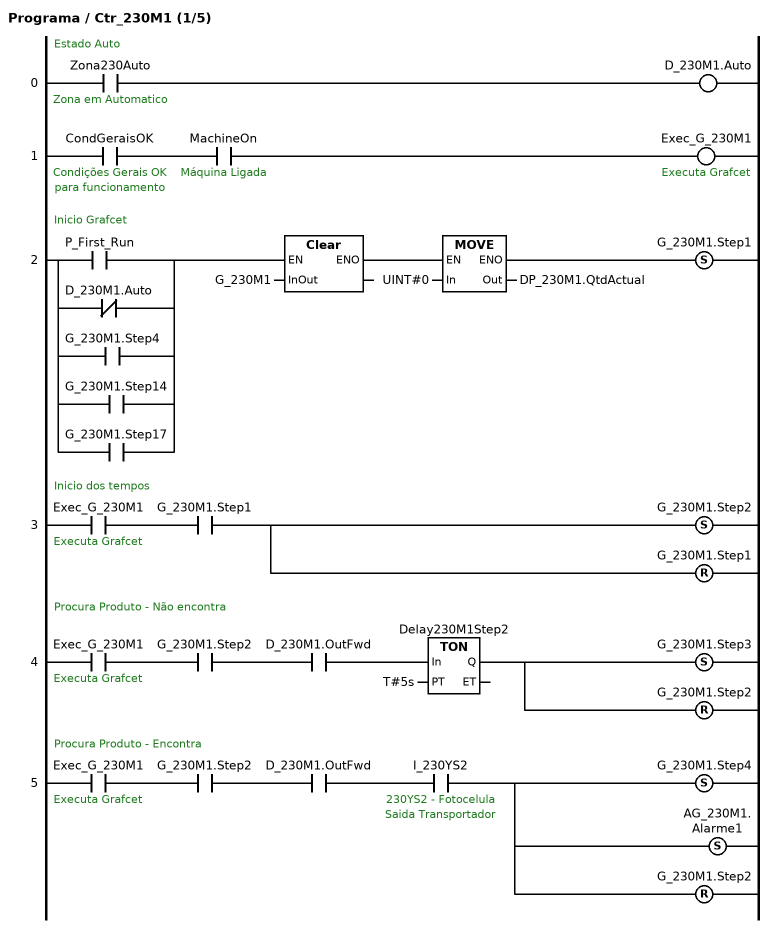
(* [picture p72: Programa / Ctr_230M1, rungs 0-5] *)
(* Rung 0: Estado Auto *)
D_230M1.Auto := Zona230Auto;
(* Rung 1 *)
Exec_G_230M1 := CondGeraisOK AND MachineOn;
(* Rung 2: Inicio Grafcet *)
_p131 := P_First_Run OR NOT D_230M1.Auto OR G_230M1.Step4 OR G_230M1.Step14 OR G_230M1.Step17;
IF _p131 THEN
    Clear(InOut := G_230M1);
    DP_230M1.QtdActual := UINT#0;
    G_230M1.Step1 := TRUE;
END_IF;
(* Rung 3: Inicio dos tempos *)
_p132 := Exec_G_230M1 AND G_230M1.Step1;
IF _p132 THEN
    G_230M1.Step2 := TRUE;
    G_230M1.Step1 := FALSE;
END_IF;
(* Rung 4: Procura Produto - Não encontra *)
Delay230M1Step2(In := Exec_G_230M1 AND G_230M1.Step2 AND D_230M1.OutFwd, PT := T#5s);
IF Delay230M1Step2.Q THEN
    G_230M1.Step3 := TRUE;
    G_230M1.Step2 := FALSE;
END_IF;
(* Rung 5: Procura Produto - Encontra *)
_p133 := Exec_G_230M1 AND G_230M1.Step2 AND D_230M1.OutFwd AND I_230YS2;
IF _p133 THEN
    G_230M1.Step4 := TRUE;
    AG_230M1.Alarme1 := TRUE;
    G_230M1.Step2 := FALSE;
END_IF;

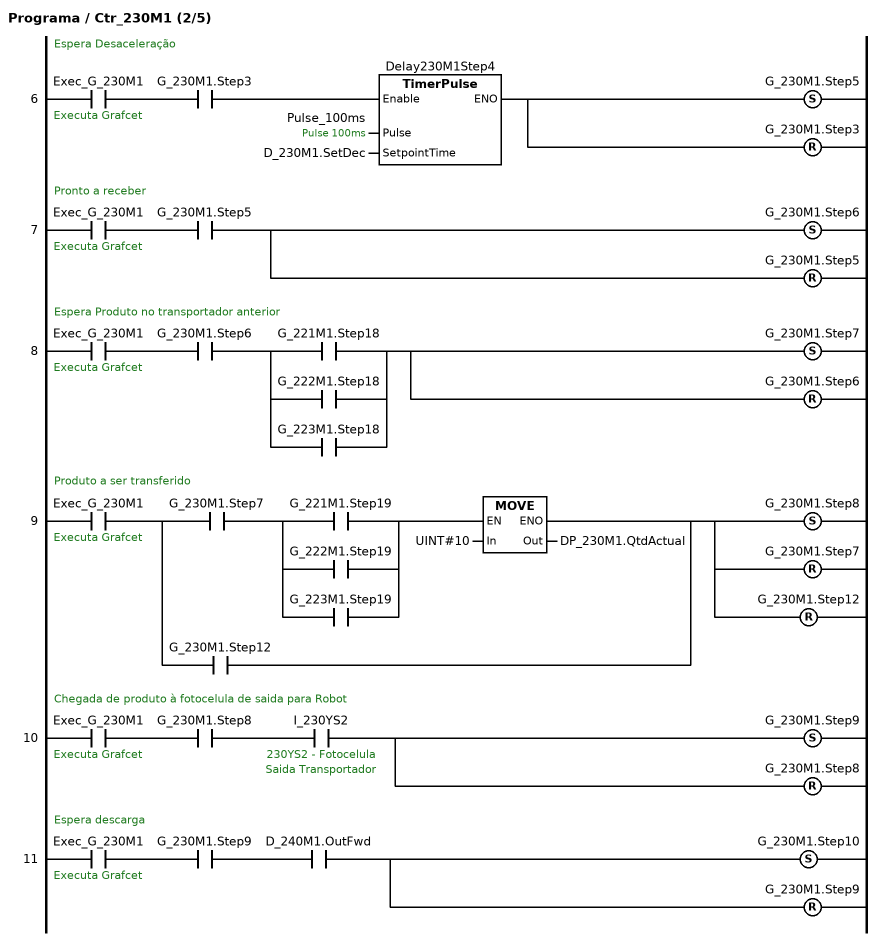
(* Rung 6: Espera Desaceleração *)
Delay230M1Step4(Enable := Exec_G_230M1 AND G_230M1.Step3, Pulse := Pulse_100ms, SetpointTime := D_230M1.SetDec);
IF Delay230M1Step4.ENO THEN
    G_230M1.Step5 := TRUE;
    G_230M1.Step3 := FALSE;
END_IF;
(* Rung 7: Pronto a receber *)
_p134 := Exec_G_230M1 AND G_230M1.Step5;
IF _p134 THEN
    G_230M1.Step6 := TRUE;
    G_230M1.Step5 := FALSE;
END_IF;
(* Rung 8: Espera Produto no transportador anterior *)
_p135 := Exec_G_230M1 AND G_230M1.Step6 AND (G_221M1.Step18 OR G_222M1.Step18 OR G_223M1.Step18);
IF _p135 THEN
    G_230M1.Step7 := TRUE;
    G_230M1.Step6 := FALSE;
END_IF;
(* Rung 9: Produto a ser transferido *)
IF Exec_G_230M1 AND G_230M1.Step7 AND (G_221M1.Step19 OR G_222M1.Step19 OR G_223M1.Step19) THEN
    DP_230M1.QtdActual := UINT#10;
END_IF;
_p136 := Exec_G_230M1 AND ((G_230M1.Step7 AND (G_221M1.Step19 OR G_222M1.Step19 OR G_223M1.Step19)) OR G_230M1.Step12);
IF _p136 THEN
    G_230M1.Step8 := TRUE;
    G_230M1.Step7 := FALSE;
    G_230M1.Step12 := FALSE;
END_IF;
(* Rung 10: Chegada de produto à fotocelula de saida para Robot *)
_p137 := Exec_G_230M1 AND G_230M1.Step8 AND I_230YS2;
IF _p137 THEN
    G_230M1.Step9 := TRUE;
    G_230M1.Step8 := FALSE;
END_IF;
(* Rung 11: Espera descarga *)
_p138 := Exec_G_230M1 AND G_230M1.Step9 AND D_240M1.OutFwd;
IF _p138 THEN
    G_230M1.Step10 := TRUE;
    G_230M1.Step9 := FALSE;
END_IF;

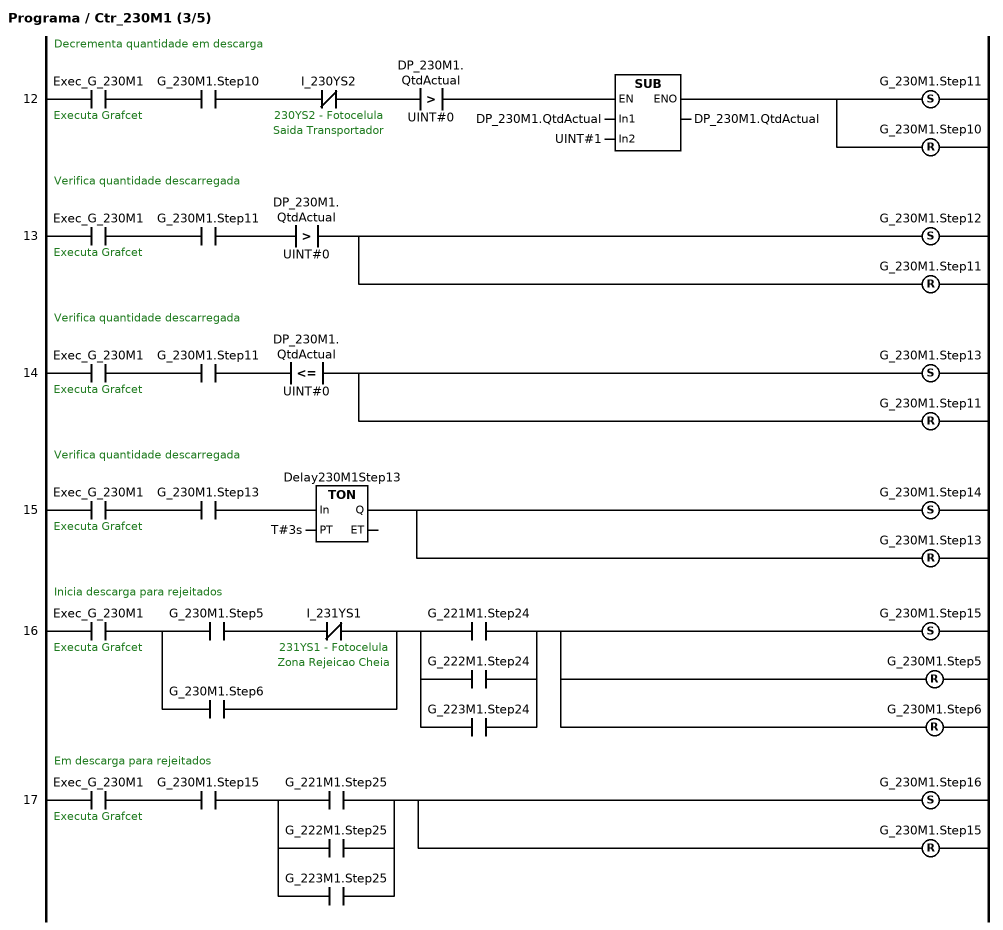
(* Rung 12: Decrementa quantidade em descarga *)
_p139 := Exec_G_230M1 AND G_230M1.Step10 AND NOT I_230YS2 AND (DP_230M1.QtdActual > UINT#0);
IF _p139 THEN
    DP_230M1.QtdActual := DP_230M1.QtdActual - UINT#1;
    G_230M1.Step11 := TRUE;
    G_230M1.Step10 := FALSE;
END_IF;
(* Rung 13: Verifica quantidade descarregada *)
_p140 := Exec_G_230M1 AND G_230M1.Step11 AND (DP_230M1.QtdActual > UINT#0);
IF _p140 THEN
    G_230M1.Step12 := TRUE;
    G_230M1.Step11 := FALSE;
END_IF;
(* Rung 14: Verifica quantidade descarregada *)
_p141 := Exec_G_230M1 AND G_230M1.Step11 AND (DP_230M1.QtdActual <= UINT#0);
IF _p141 THEN
    G_230M1.Step13 := TRUE;
    G_230M1.Step11 := FALSE;
END_IF;
(* Rung 15: Verifica quantidade descarregada *)
Delay230M1Step13(In := Exec_G_230M1 AND G_230M1.Step13, PT := T#3s);
IF Delay230M1Step13.Q THEN
    G_230M1.Step14 := TRUE;
    G_230M1.Step13 := FALSE;
END_IF;
(* Rung 16: Inicia descarga para rejeitados *)
_p142 := Exec_G_230M1 AND ((G_230M1.Step5 AND NOT I_231YS1) OR G_230M1.Step6) AND (G_221M1.Step24 OR G_222M1.Step24 OR G_223M1.Step24);
IF _p142 THEN
    G_230M1.Step15 := TRUE;
    G_230M1.Step5 := FALSE;
    G_230M1.Step6 := FALSE;
END_IF;
(* Rung 17: Em descarga para rejeitados *)
_p143 := Exec_G_230M1 AND G_230M1.Step15 AND (G_221M1.Step25 OR G_222M1.Step25 OR G_223M1.Step25);
IF _p143 THEN
    G_230M1.Step16 := TRUE;
    G_230M1.Step15 := FALSE;
END_IF;

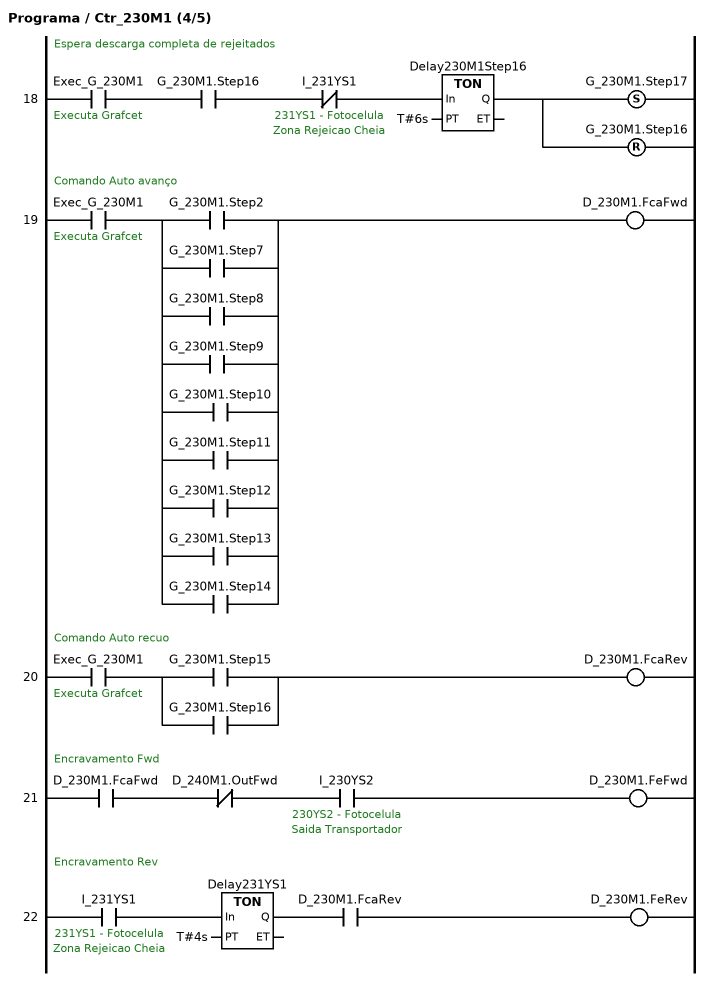
(* Rung 18: Espera descarga completa de rejeitados *)
Delay230M1Step16(In := Exec_G_230M1 AND G_230M1.Step16 AND NOT I_231YS1, PT := T#6s);
IF Delay230M1Step16.Q THEN
    G_230M1.Step17 := TRUE;
    G_230M1.Step16 := FALSE;
END_IF;
(* Rung 19: Comando Auto avanço *)
D_230M1.FcaFwd := Exec_G_230M1 AND (G_230M1.Step2 OR G_230M1.Step7 OR G_230M1.Step8 OR G_230M1.Step9 OR G_230M1.Step10 OR G_230M1.Step11 OR G_230M1.Step12 OR G_230M1.Step13 OR G_230M1.Step14);
(* Rung 20: Comando Auto recuo *)
D_230M1.FcaRev := Exec_G_230M1 AND (G_230M1.Step15 OR G_230M1.Step16);
(* Rung 21: Encravamento Fwd *)
D_230M1.FeFwd := D_230M1.FcaFwd AND NOT D_240M1.OutFwd AND I_230YS2;
(* Rung 22: Encravamento Rev *)
Delay231YS1(In := I_231YS1, PT := T#4s);
D_230M1.FeRev := Delay231YS1.Q AND D_230M1.FcaRev;

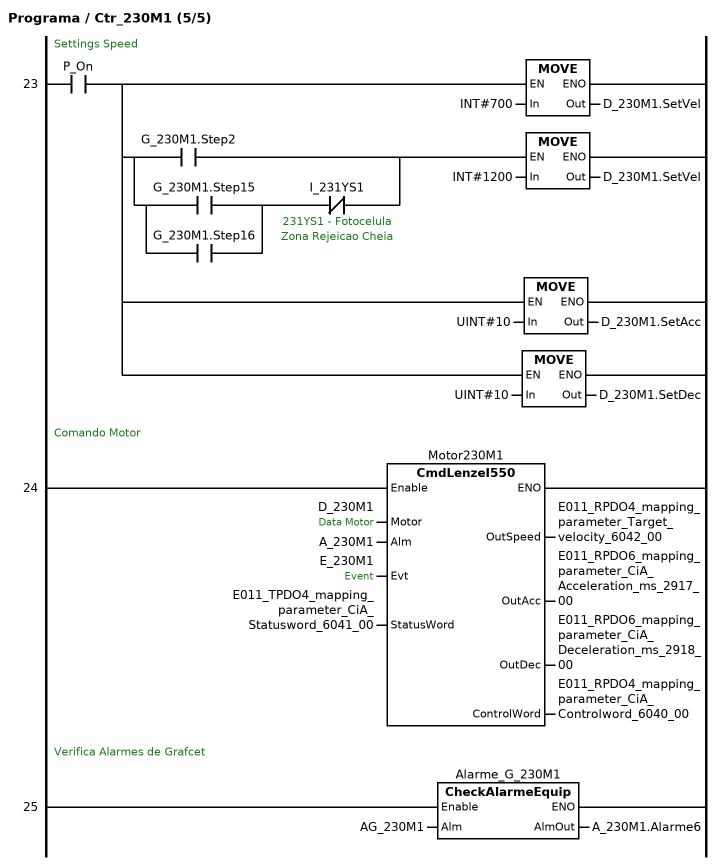
(* Rung 23: Settings Speed *)
IF P_On THEN D_230M1.SetVel := INT#700; END_IF;
IF P_On AND (G_230M1.Step2 OR ((G_230M1.Step15 OR G_230M1.Step16) AND NOT I_231YS1)) THEN
    D_230M1.SetVel := INT#1200;
END_IF;
IF P_On THEN
    D_230M1.SetAcc := UINT#10;
    D_230M1.SetDec := UINT#10;
END_IF;
(* Rung 24: Comando Motor *)
Motor230M1(Enable := TRUE, Motor := D_230M1, Alm := A_230M1, Evt := E_230M1, StatusWord := E011_TPDO4_mapping_parameter_CiA_Statusword_6041_00, OutSpeed => E011_RPDO4_mapping_parameter_Target_velocity_6042_00, OutAcc => E011_RPDO6_mapping_parameter_CiA_Acceleration_ms_2917_00, OutDec => E011_RPDO6_mapping_parameter_CiA_Deceleration_ms_2918_00, ControlWord => E011_RPDO4_mapping_parameter_CiA_Controlword_6040_00);
(* Rung 25: Verifica Alarmes de Grafcet *)
Alarme_G_230M1(Enable := TRUE, Alm := AG_230M1, AlmOut => A_230M1.Alarme6);

(* Section Ctr_240M1: ladder, written here as Structured Text *)

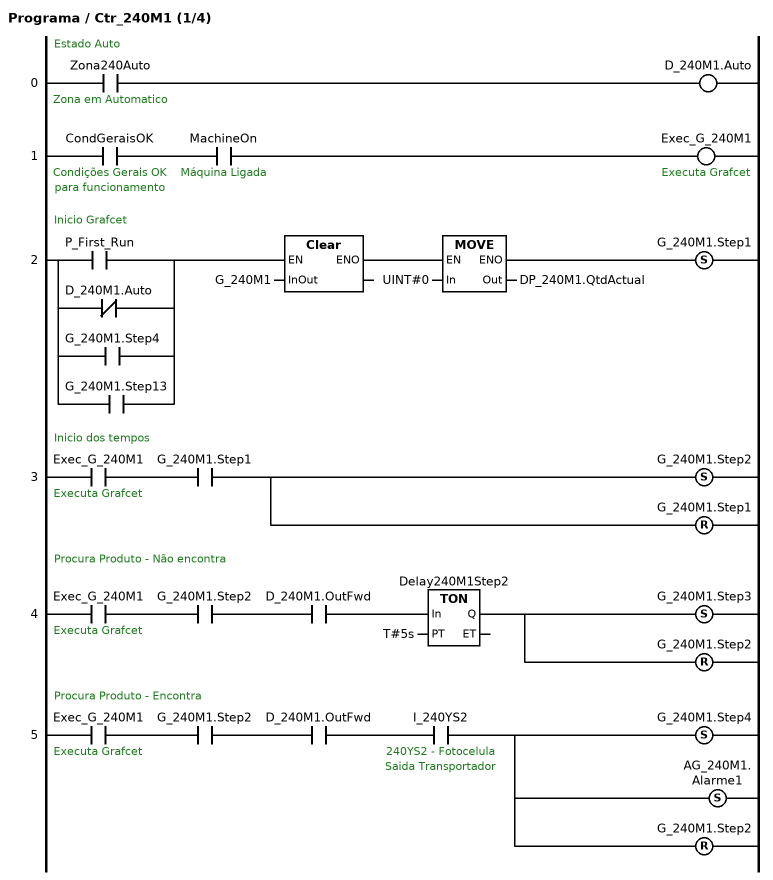
(* Rung 0: Estado Auto *)
D_240M1.Auto := Zona240Auto;
(* Rung 1 *)
Exec_G_240M1 := CondGeraisOK AND MachineOn;
(* Rung 2: Inicio Grafcet *)
_p144 := P_First_Run OR NOT D_240M1.Auto OR G_240M1.Step4 OR G_240M1.Step13;
IF _p144 THEN
    Clear(InOut := G_240M1);
    DP_240M1.QtdActual := UINT#0;
    G_240M1.Step1 := TRUE;
END_IF;
(* Rung 3: Inicio dos tempos *)
_p145 := Exec_G_240M1 AND G_240M1.Step1;
IF _p145 THEN
    G_240M1.Step2 := TRUE;
    G_240M1.Step1 := FALSE;
END_IF;
(* Rung 4: Procura Produto - Não encontra *)
Delay240M1Step2(In := Exec_G_240M1 AND G_240M1.Step2 AND D_240M1.OutFwd, PT := T#5s);
IF Delay240M1Step2.Q THEN
    G_240M1.Step3 := TRUE;
    G_240M1.Step2 := FALSE;
END_IF;
(* Rung 5: Procura Produto - Encontra *)
_p146 := Exec_G_240M1 AND G_240M1.Step2 AND D_240M1.OutFwd AND I_240YS2;
IF _p146 THEN
    G_240M1.Step4 := TRUE;
    AG_240M1.Alarme1 := TRUE;
    G_240M1.Step2 := FALSE;
END_IF;

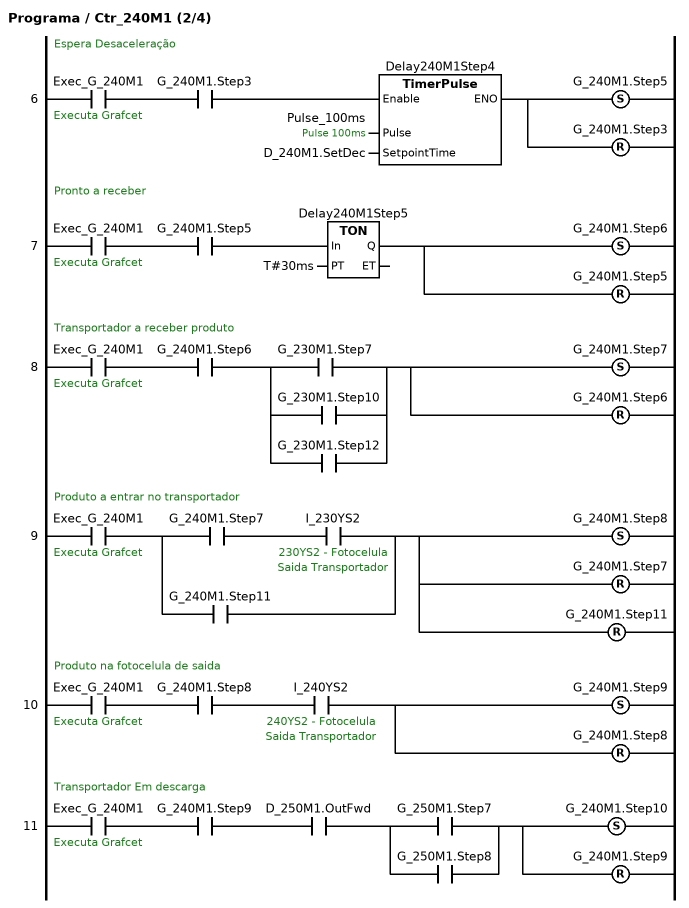
(* Rung 6: Espera Desaceleração *)
Delay240M1Step4(Enable := Exec_G_240M1 AND G_240M1.Step3, Pulse := Pulse_100ms, SetpointTime := D_240M1.SetDec);
IF Delay240M1Step4.ENO THEN
    G_240M1.Step5 := TRUE;
    G_240M1.Step3 := FALSE;
END_IF;
(* Rung 7: Pronto a receber *)
Delay240M1Step5(In := Exec_G_240M1 AND G_240M1.Step5, PT := T#30ms);
IF Delay240M1Step5.Q THEN
    G_240M1.Step6 := TRUE;
    G_240M1.Step5 := FALSE;
END_IF;
(* Rung 8: Transportador a receber produto *)
_p147 := Exec_G_240M1 AND G_240M1.Step6 AND (G_230M1.Step7 OR G_230M1.Step10 OR G_230M1.Step12);
IF _p147 THEN
    G_240M1.Step7 := TRUE;
    G_240M1.Step6 := FALSE;
END_IF;
(* Rung 9: Produto a entrar no transportador *)
_p148 := Exec_G_240M1 AND ((G_240M1.Step7 AND I_230YS2) OR G_240M1.Step11);
IF _p148 THEN
    G_240M1.Step8 := TRUE;
    G_240M1.Step7 := FALSE;
    G_240M1.Step11 := FALSE;
END_IF;
(* Rung 10: Produto na fotocelula de saida *)
_p149 := Exec_G_240M1 AND G_240M1.Step8 AND I_240YS2;
IF _p149 THEN
    G_240M1.Step9 := TRUE;
    G_240M1.Step8 := FALSE;
END_IF;
(* Rung 11: Transportador Em descarga *)
_p150 := Exec_G_240M1 AND G_240M1.Step9 AND D_250M1.OutFwd AND (G_250M1.Step7 OR G_250M1.Step8);
IF _p150 THEN
    G_240M1.Step10 := TRUE;
    G_240M1.Step9 := FALSE;
END_IF;

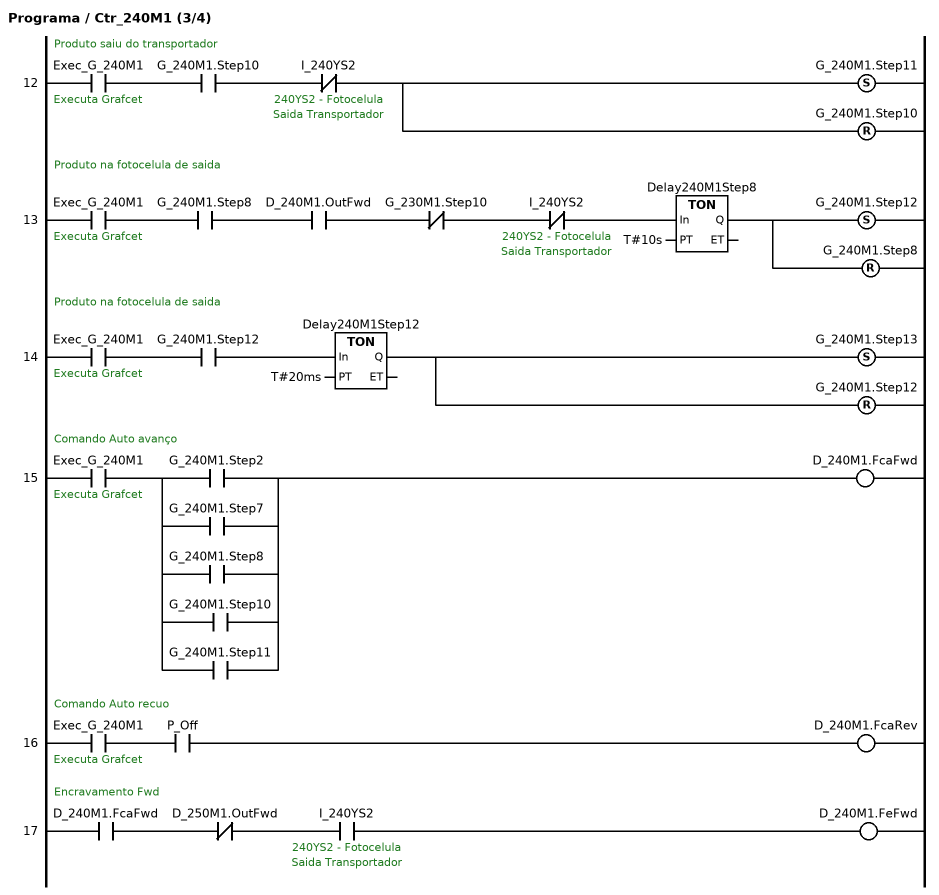
(* Rung 12: Produto saiu do transportador *)
_p151 := Exec_G_240M1 AND G_240M1.Step10 AND NOT I_240YS2;
IF _p151 THEN
    G_240M1.Step11 := TRUE;
    G_240M1.Step10 := FALSE;
END_IF;
(* Rung 13: Produto na fotocelula de saida *)
Delay240M1Step8(In := Exec_G_240M1 AND G_240M1.Step8 AND D_240M1.OutFwd AND NOT G_230M1.Step10 AND NOT I_240YS2, PT := T#10s);
IF Delay240M1Step8.Q THEN
    G_240M1.Step12 := TRUE;
    G_240M1.Step8 := FALSE;
END_IF;
(* Rung 14: Produto na fotocelula de saida *)
Delay240M1Step12(In := Exec_G_240M1 AND G_240M1.Step12, PT := T#20ms);
IF Delay240M1Step12.Q THEN
    G_240M1.Step13 := TRUE;
    G_240M1.Step12 := FALSE;
END_IF;
(* Rung 15: Comando Auto avanço *)
D_240M1.FcaFwd := Exec_G_240M1 AND (G_240M1.Step2 OR G_240M1.Step7 OR G_240M1.Step8 OR G_240M1.Step10 OR G_240M1.Step11);
(* Rung 16: Comando Auto recuo *)
D_240M1.FcaRev := Exec_G_240M1 AND P_Off;
(* Rung 17: Encravamento Fwd *)
D_240M1.FeFwd := D_240M1.FcaFwd AND NOT D_250M1.OutFwd AND I_240YS2;

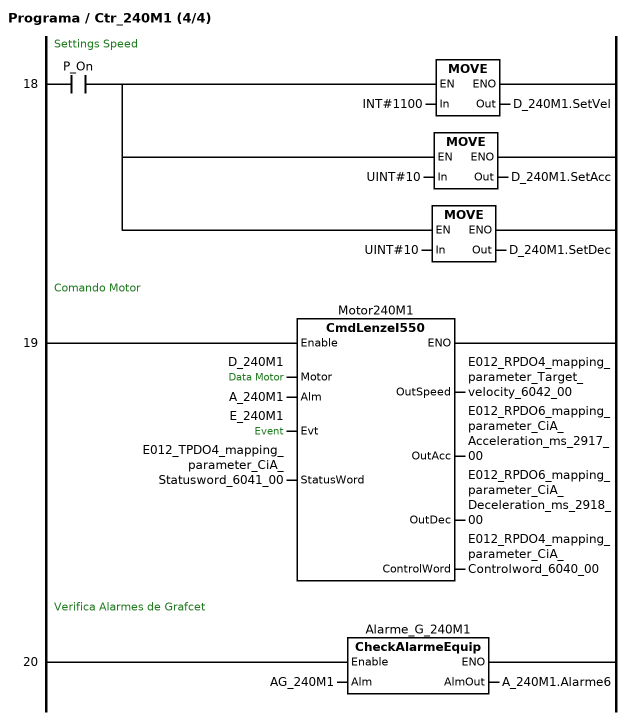
(* Rung 18: Settings Speed *)
IF P_On THEN
    D_240M1.SetVel := INT#1100;
    D_240M1.SetAcc := UINT#10;
    D_240M1.SetDec := UINT#10;
END_IF;
(* Rung 19: Comando Motor *)
Motor240M1(Enable := TRUE, Motor := D_240M1, Alm := A_240M1, Evt := E_240M1, StatusWord := E012_TPDO4_mapping_parameter_CiA_Statusword_6041_00, OutSpeed => E012_RPDO4_mapping_parameter_Target_velocity_6042_00, OutAcc => E012_RPDO6_mapping_parameter_CiA_Acceleration_ms_2917_00, OutDec => E012_RPDO6_mapping_parameter_CiA_Deceleration_ms_2918_00, ControlWord => E012_RPDO4_mapping_parameter_CiA_Controlword_6040_00);
(* Rung 20: Verifica Alarmes de Grafcet *)
Alarme_G_240M1(Enable := TRUE, Alm := AG_240M1, AlmOut => A_240M1.Alarme6);

(* Section Ctr_250M1: ladder, written here as Structured Text *)

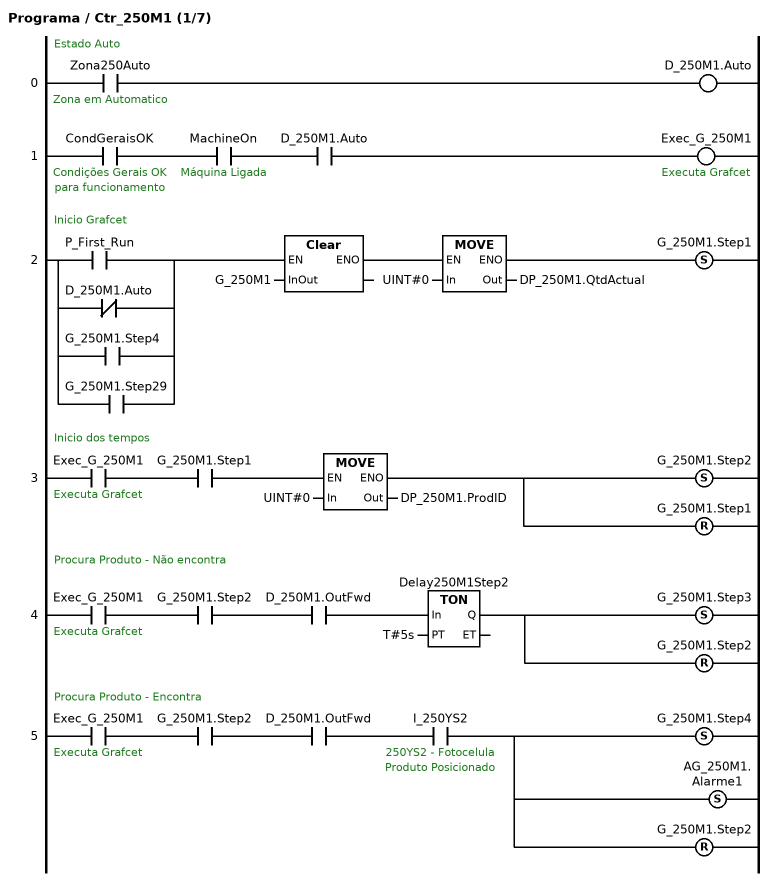
(* Rung 0: Estado Auto *)
D_250M1.Auto := Zona250Auto;
(* Rung 1 *)
Exec_G_250M1 := CondGeraisOK AND MachineOn AND D_250M1.Auto;
(* Rung 2: Inicio Grafcet *)
_p152 := P_First_Run OR NOT D_250M1.Auto OR G_250M1.Step4 OR G_250M1.Step29;
IF _p152 THEN
    Clear(InOut := G_250M1);
    DP_250M1.QtdActual := UINT#0;
    G_250M1.Step1 := TRUE;
END_IF;
(* Rung 3: Inicio dos tempos *)
IF Exec_G_250M1 AND G_250M1.Step1 THEN DP_250M1.ProdID := UINT#0; END_IF;
_p153 := Exec_G_250M1 AND G_250M1.Step1;
IF _p153 THEN
    G_250M1.Step2 := TRUE;
    G_250M1.Step1 := FALSE;
END_IF;
(* Rung 4: Procura Produto - Não encontra *)
Delay250M1Step2(In := Exec_G_250M1 AND G_250M1.Step2 AND D_250M1.OutFwd, PT := T#5s);
IF Delay250M1Step2.Q THEN
    G_250M1.Step3 := TRUE;
    G_250M1.Step2 := FALSE;
END_IF;
(* Rung 5: Procura Produto - Encontra *)
_p154 := Exec_G_250M1 AND G_250M1.Step2 AND D_250M1.OutFwd AND I_250YS2;
IF _p154 THEN
    G_250M1.Step4 := TRUE;
    AG_250M1.Alarme1 := TRUE;
    G_250M1.Step2 := FALSE;
END_IF;

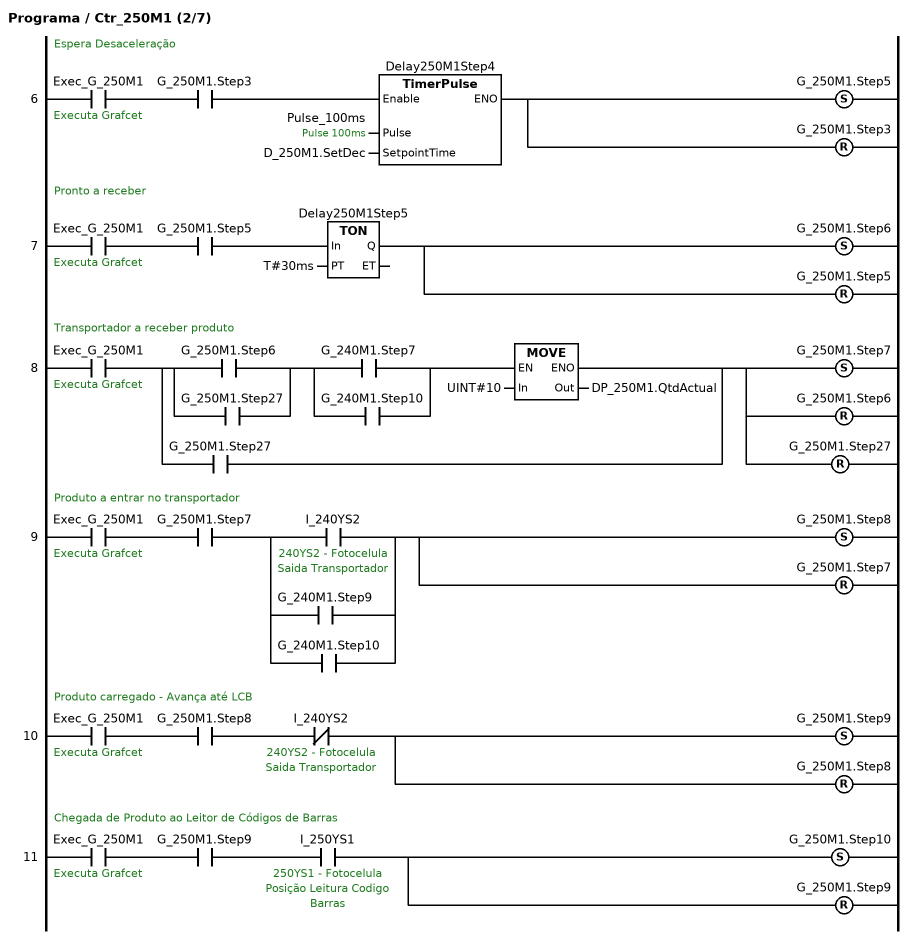
(* Rung 6: Espera Desaceleração *)
Delay250M1Step4(Enable := Exec_G_250M1 AND G_250M1.Step3, Pulse := Pulse_100ms, SetpointTime := D_250M1.SetDec);
IF Delay250M1Step4.ENO THEN
    G_250M1.Step5 := TRUE;
    G_250M1.Step3 := FALSE;
END_IF;
(* Rung 7: Pronto a receber *)
Delay250M1Step5(In := Exec_G_250M1 AND G_250M1.Step5, PT := T#30ms);
IF Delay250M1Step5.Q THEN
    G_250M1.Step6 := TRUE;
    G_250M1.Step5 := FALSE;
END_IF;
(* Rung 8: Transportador a receber produto *)
IF Exec_G_250M1 AND (G_250M1.Step6 OR G_250M1.Step27) AND (G_240M1.Step7 OR G_240M1.Step10) THEN
    DP_250M1.QtdActual := UINT#10;
END_IF;
_p155 := Exec_G_250M1 AND (((G_250M1.Step6 OR G_250M1.Step27) AND (G_240M1.Step7 OR G_240M1.Step10)) OR G_250M1.Step27);
IF _p155 THEN
    G_250M1.Step7 := TRUE;
    G_250M1.Step6 := FALSE;
    G_250M1.Step27 := FALSE;
END_IF;
(* Rung 9: Produto a entrar no transportador *)
_p156 := Exec_G_250M1 AND G_250M1.Step7 AND (I_240YS2 OR G_240M1.Step9 OR G_240M1.Step10);
IF _p156 THEN
    G_250M1.Step8 := TRUE;
    G_250M1.Step7 := FALSE;
END_IF;
(* Rung 10: Produto carregado - Avança até LCB *)
_p157 := Exec_G_250M1 AND G_250M1.Step8 AND NOT I_240YS2;
IF _p157 THEN
    G_250M1.Step9 := TRUE;
    G_250M1.Step8 := FALSE;
END_IF;
(* Rung 11: Chegada de Produto ao Leitor de Códigos de Barras *)
_p158 := Exec_G_250M1 AND G_250M1.Step9 AND I_250YS1;
IF _p158 THEN
    G_250M1.Step10 := TRUE;
    G_250M1.Step9 := FALSE;
END_IF;

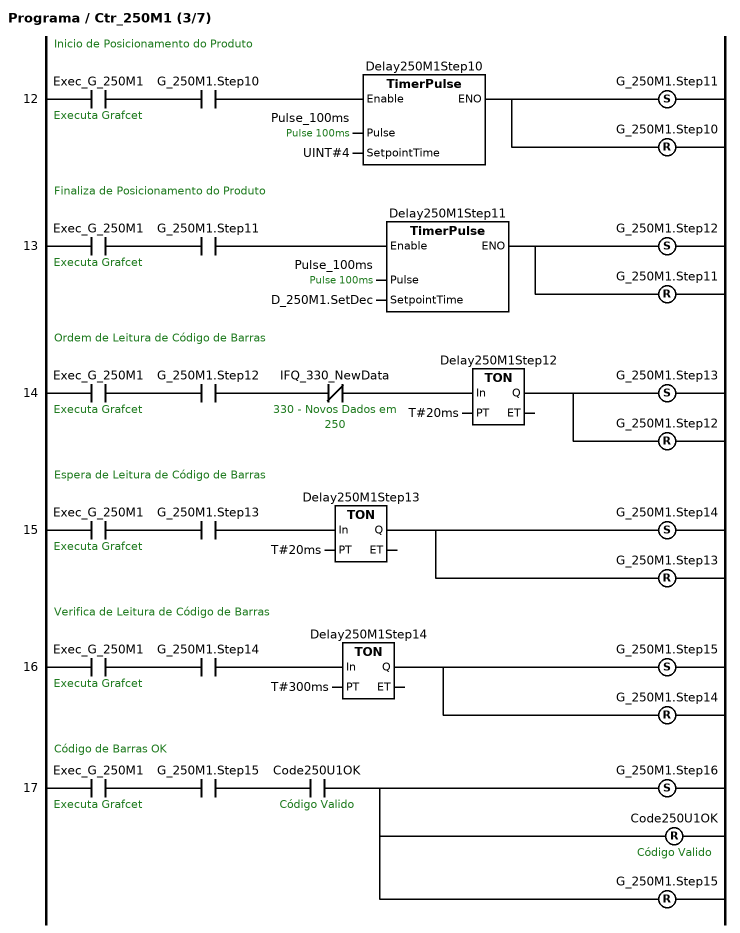
(* Rung 12: Inicio de Posicionamento do Produto *)
Delay250M1Step10(Enable := Exec_G_250M1 AND G_250M1.Step10, Pulse := Pulse_100ms, SetpointTime := UINT#4);
IF Delay250M1Step10.ENO THEN
    G_250M1.Step11 := TRUE;
    G_250M1.Step10 := FALSE;
END_IF;
(* Rung 13: Finaliza de Posicionamento do Produto *)
Delay250M1Step11(Enable := Exec_G_250M1 AND G_250M1.Step11, Pulse := Pulse_100ms, SetpointTime := D_250M1.SetDec);
IF Delay250M1Step11.ENO THEN
    G_250M1.Step12 := TRUE;
    G_250M1.Step11 := FALSE;
END_IF;
(* Rung 14: Ordem de Leitura de Código de Barras *)
Delay250M1Step12(In := Exec_G_250M1 AND G_250M1.Step12 AND NOT IFQ_330_NewData, PT := T#20ms);
IF Delay250M1Step12.Q THEN
    G_250M1.Step13 := TRUE;
    G_250M1.Step12 := FALSE;
END_IF;
(* Rung 15: Espera de Leitura de Código de Barras *)
Delay250M1Step13(In := Exec_G_250M1 AND G_250M1.Step13, PT := T#20ms);
IF Delay250M1Step13.Q THEN
    G_250M1.Step14 := TRUE;
    G_250M1.Step13 := FALSE;
END_IF;
(* Rung 16: Verifica de Leitura de Código de Barras *)
Delay250M1Step14(In := Exec_G_250M1 AND G_250M1.Step14, PT := T#300ms);
IF Delay250M1Step14.Q THEN
    G_250M1.Step15 := TRUE;
    G_250M1.Step14 := FALSE;
END_IF;
(* Rung 17: Código de Barras OK *)
_p159 := Exec_G_250M1 AND G_250M1.Step15 AND Code250U1OK;
IF _p159 THEN
    G_250M1.Step16 := TRUE;
    Code250U1OK := FALSE;
    G_250M1.Step15 := FALSE;
END_IF;

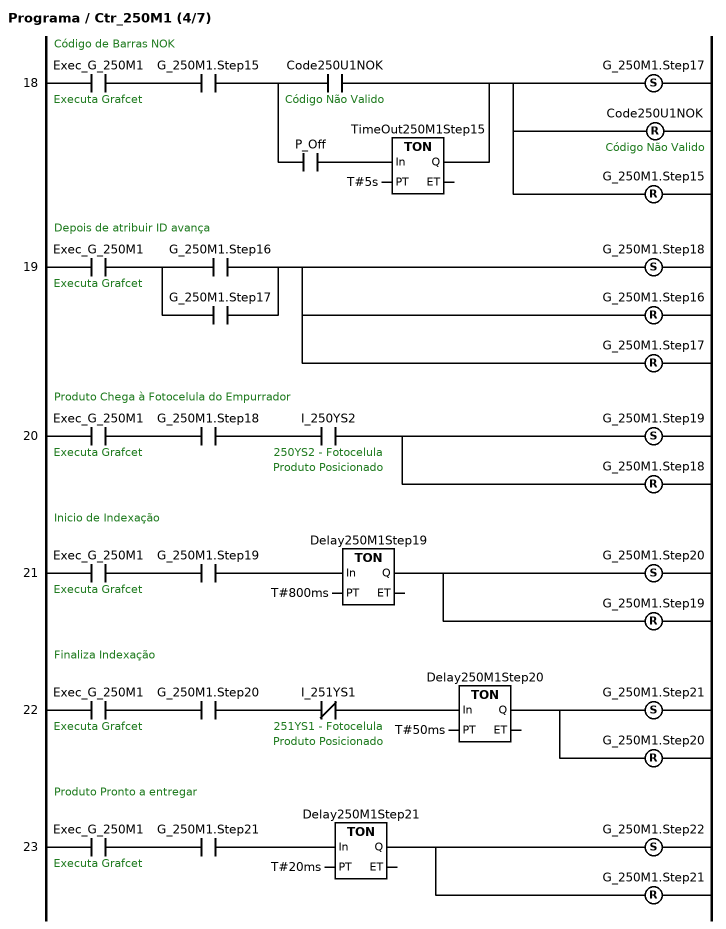
(* Rung 18: Código de Barras NOK *)
TimeOut250M1Step15(In := Exec_G_250M1 AND G_250M1.Step15 AND P_Off, PT := T#5s);
_p160 := (Exec_G_250M1 AND G_250M1.Step15 AND Code250U1NOK) OR TimeOut250M1Step15.Q;
IF _p160 THEN
    G_250M1.Step17 := TRUE;
    Code250U1NOK := FALSE;
    G_250M1.Step15 := FALSE;
END_IF;
(* Rung 19: Depois de atribuir ID avança *)
_p161 := Exec_G_250M1 AND (G_250M1.Step16 OR G_250M1.Step17);
IF _p161 THEN
    G_250M1.Step18 := TRUE;
    G_250M1.Step16 := FALSE;
    G_250M1.Step17 := FALSE;
END_IF;
(* Rung 20: Produto Chega à Fotocelula do Empurrador *)
_p162 := Exec_G_250M1 AND G_250M1.Step18 AND I_250YS2;
IF _p162 THEN
    G_250M1.Step19 := TRUE;
    G_250M1.Step18 := FALSE;
END_IF;
(* Rung 21: Inicio de Indexação *)
Delay250M1Step19(In := Exec_G_250M1 AND G_250M1.Step19, PT := T#800ms);
IF Delay250M1Step19.Q THEN
    G_250M1.Step20 := TRUE;
    G_250M1.Step19 := FALSE;
END_IF;
(* Rung 22: Finaliza Indexação *)
Delay250M1Step20(In := Exec_G_250M1 AND G_250M1.Step20 AND NOT I_251YS1, PT := T#50ms);
IF Delay250M1Step20.Q THEN
    G_250M1.Step21 := TRUE;
    G_250M1.Step20 := FALSE;
END_IF;
(* Rung 23: Produto Pronto a entregar *)
Delay250M1Step21(In := Exec_G_250M1 AND G_250M1.Step21, PT := T#20ms);
IF Delay250M1Step21.Q THEN
    G_250M1.Step22 := TRUE;
    G_250M1.Step21 := FALSE;
END_IF;

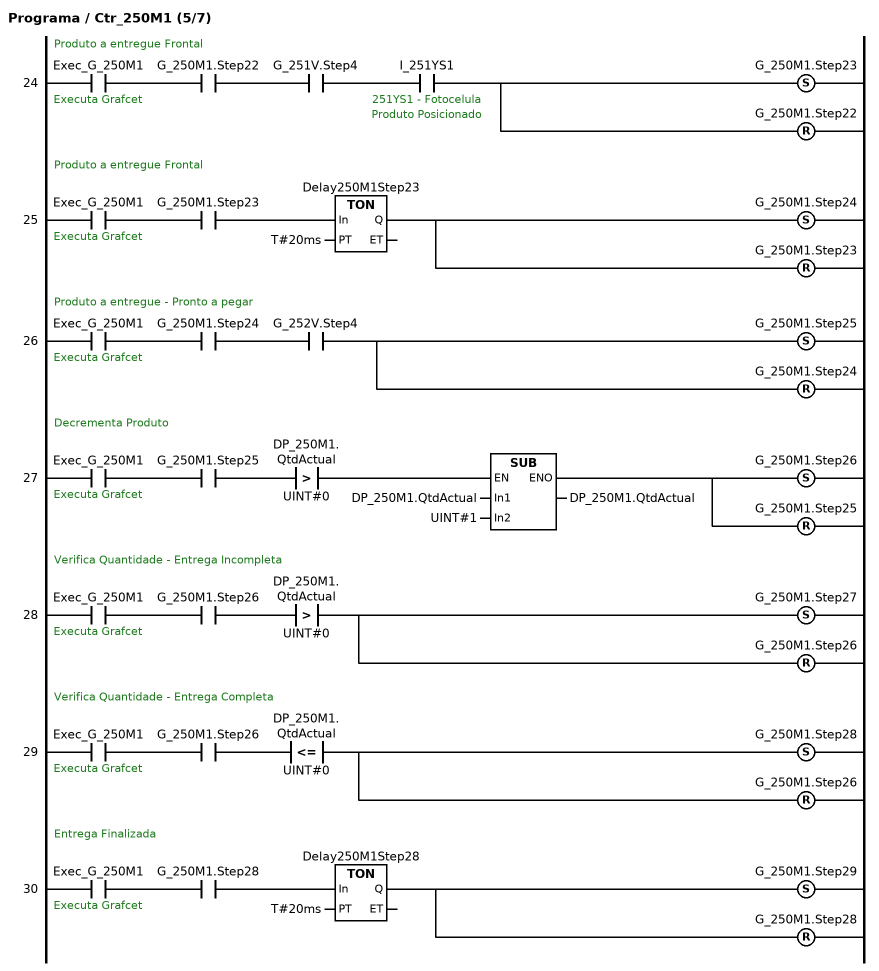
(* Rung 24: Produto a entregue Frontal *)
_p163 := Exec_G_250M1 AND G_250M1.Step22 AND G_251V.Step4 AND I_251YS1;
IF _p163 THEN
    G_250M1.Step23 := TRUE;
    G_250M1.Step22 := FALSE;
END_IF;
(* Rung 25: Produto a entregue Frontal *)
Delay250M1Step23(In := Exec_G_250M1 AND G_250M1.Step23, PT := T#20ms);
IF Delay250M1Step23.Q THEN
    G_250M1.Step24 := TRUE;
    G_250M1.Step23 := FALSE;
END_IF;
(* Rung 26: Produto a entregue - Pronto a pegar *)
_p164 := Exec_G_250M1 AND G_250M1.Step24 AND G_252V.Step4;
IF _p164 THEN
    G_250M1.Step25 := TRUE;
    G_250M1.Step24 := FALSE;
END_IF;
(* Rung 27: Decrementa Produto *)
_p165 := Exec_G_250M1 AND G_250M1.Step25 AND (DP_250M1.QtdActual > UINT#0);
IF _p165 THEN
    DP_250M1.QtdActual := DP_250M1.QtdActual - UINT#1;
    G_250M1.Step26 := TRUE;
    G_250M1.Step25 := FALSE;
END_IF;
(* Rung 28: Verifica Quantidade - Entrega Incompleta *)
_p166 := Exec_G_250M1 AND G_250M1.Step26 AND (DP_250M1.QtdActual > UINT#0);
IF _p166 THEN
    G_250M1.Step27 := TRUE;
    G_250M1.Step26 := FALSE;
END_IF;
(* Rung 29: Verifica Quantidade - Entrega Completa *)
_p167 := Exec_G_250M1 AND G_250M1.Step26 AND (DP_250M1.QtdActual <= UINT#0);
IF _p167 THEN
    G_250M1.Step28 := TRUE;
    G_250M1.Step26 := FALSE;
END_IF;
(* Rung 30: Entrega Finalizada *)
Delay250M1Step28(In := Exec_G_250M1 AND G_250M1.Step28, PT := T#20ms);
IF Delay250M1Step28.Q THEN
    G_250M1.Step29 := TRUE;
    G_250M1.Step28 := FALSE;
END_IF;

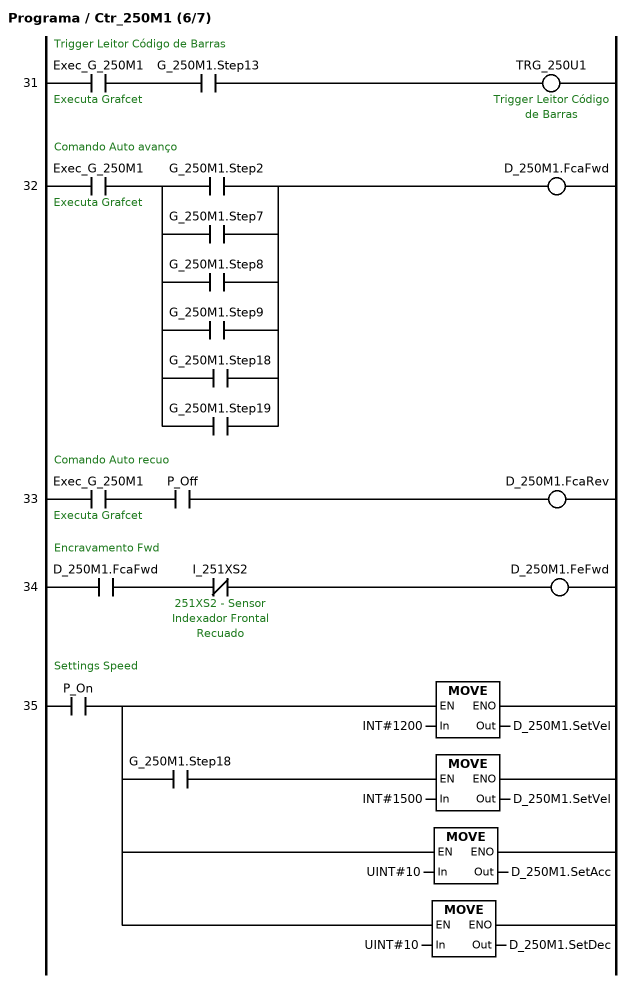
(* Rung 31: Trigger Leitor Código de Barras *)
TRG_250U1 := Exec_G_250M1 AND G_250M1.Step13;
(* Rung 32: Comando Auto avanço *)
D_250M1.FcaFwd := Exec_G_250M1 AND (G_250M1.Step2 OR G_250M1.Step7 OR G_250M1.Step8 OR G_250M1.Step9 OR G_250M1.Step18 OR G_250M1.Step19);
(* Rung 33: Comando Auto recuo *)
D_250M1.FcaRev := Exec_G_250M1 AND P_Off;
(* Rung 34: Encravamento Fwd *)
D_250M1.FeFwd := D_250M1.FcaFwd AND NOT I_251XS2;
(* Rung 35: Settings Speed *)
IF P_On THEN D_250M1.SetVel := INT#1200; END_IF;
IF P_On AND G_250M1.Step18 THEN D_250M1.SetVel := INT#1500; END_IF;
IF P_On THEN
    D_250M1.SetAcc := UINT#10;
    D_250M1.SetDec := UINT#10;
END_IF;

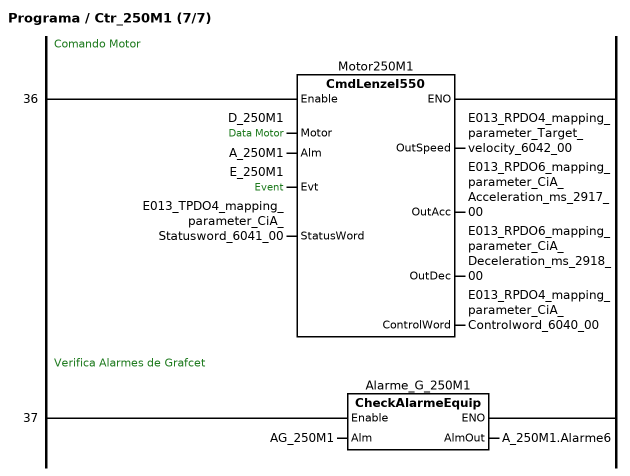
(* Rung 36: Comando Motor *)
Motor250M1(Enable := TRUE, Motor := D_250M1, Alm := A_250M1, Evt := E_250M1, StatusWord := E013_TPDO4_mapping_parameter_CiA_Statusword_6041_00, OutSpeed => E013_RPDO4_mapping_parameter_Target_velocity_6042_00, OutAcc => E013_RPDO6_mapping_parameter_CiA_Acceleration_ms_2917_00, OutDec => E013_RPDO6_mapping_parameter_CiA_Deceleration_ms_2918_00, ControlWord => E013_RPDO4_mapping_parameter_CiA_Controlword_6040_00);
(* Rung 37: Verifica Alarmes de Grafcet *)
Alarme_G_250M1(Enable := TRUE, Alm := AG_250M1, AlmOut => A_250M1.Alarme6);

(* Section Data_250U1: ladder, written here as Structured Text *)

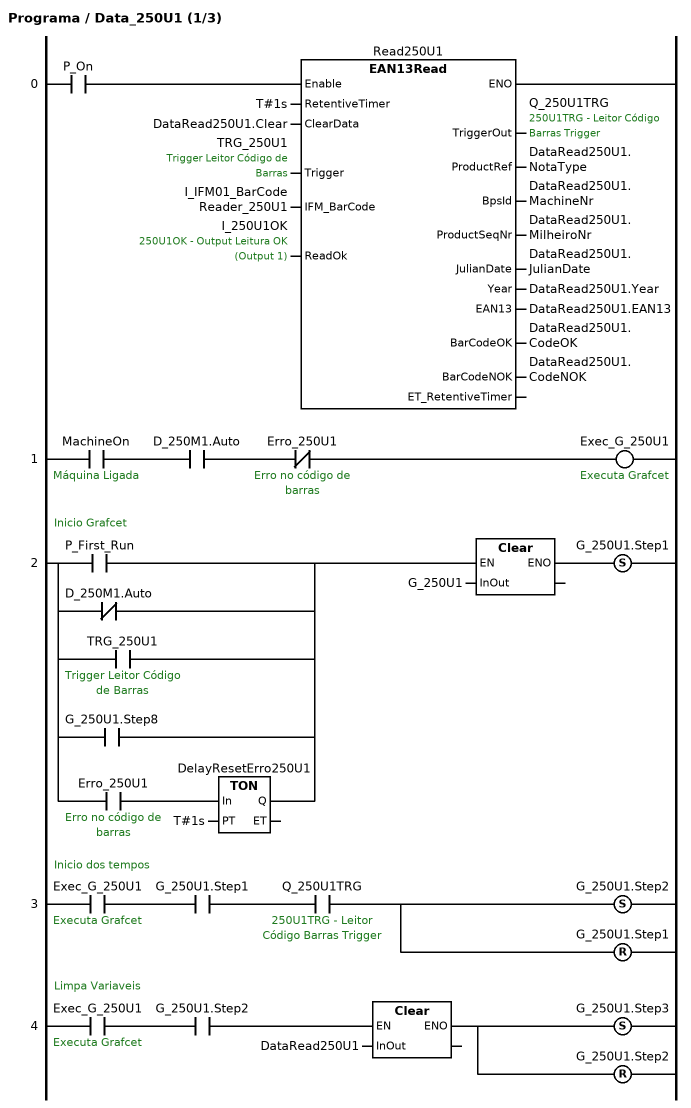
(* Rung 0 *)
Read250U1(Enable := P_On, RetentiveTimer := T#1s, ClearData := DataRead250U1.Clear, Trigger := TRG_250U1, IFM_BarCode := I_IFM01_BarCodeReader_250U1, ReadOk := I_250U1OK, TriggerOut => Q_250U1TRG, ProductRef => DataRead250U1.NotaType, BpsId => DataRead250U1.MachineNr, ProductSeqNr => DataRead250U1.MilheiroNr, JulianDate => DataRead250U1.JulianDate, Year => DataRead250U1.Year, EAN13 => DataRead250U1.EAN13, BarCodeOK => DataRead250U1.CodeOK, BarCodeNOK => DataRead250U1.CodeNOK);
(* Rung 1 *)
Exec_G_250U1 := MachineOn AND D_250M1.Auto AND NOT Erro_250U1;
(* Rung 2: Inicio Grafcet *)
DelayResetErro250U1(In := Erro_250U1, PT := T#1s);
_p168 := P_First_Run OR NOT D_250M1.Auto OR TRG_250U1 OR G_250U1.Step8 OR DelayResetErro250U1.Q;
IF _p168 THEN
    Clear(InOut := G_250U1);
    G_250U1.Step1 := TRUE;
END_IF;
(* Rung 3: Inicio dos tempos *)
_p169 := Exec_G_250U1 AND G_250U1.Step1 AND Q_250U1TRG;
IF _p169 THEN
    G_250U1.Step2 := TRUE;
    G_250U1.Step1 := FALSE;
END_IF;
(* Rung 4: Limpa Variaveis *)
IF Exec_G_250U1 AND G_250U1.Step2 THEN Clear(InOut := DataRead250U1); END_IF;
_p170 := Exec_G_250U1 AND G_250U1.Step2;
IF _p170 THEN
    G_250U1.Step3 := TRUE;
    G_250U1.Step2 := FALSE;
END_IF;

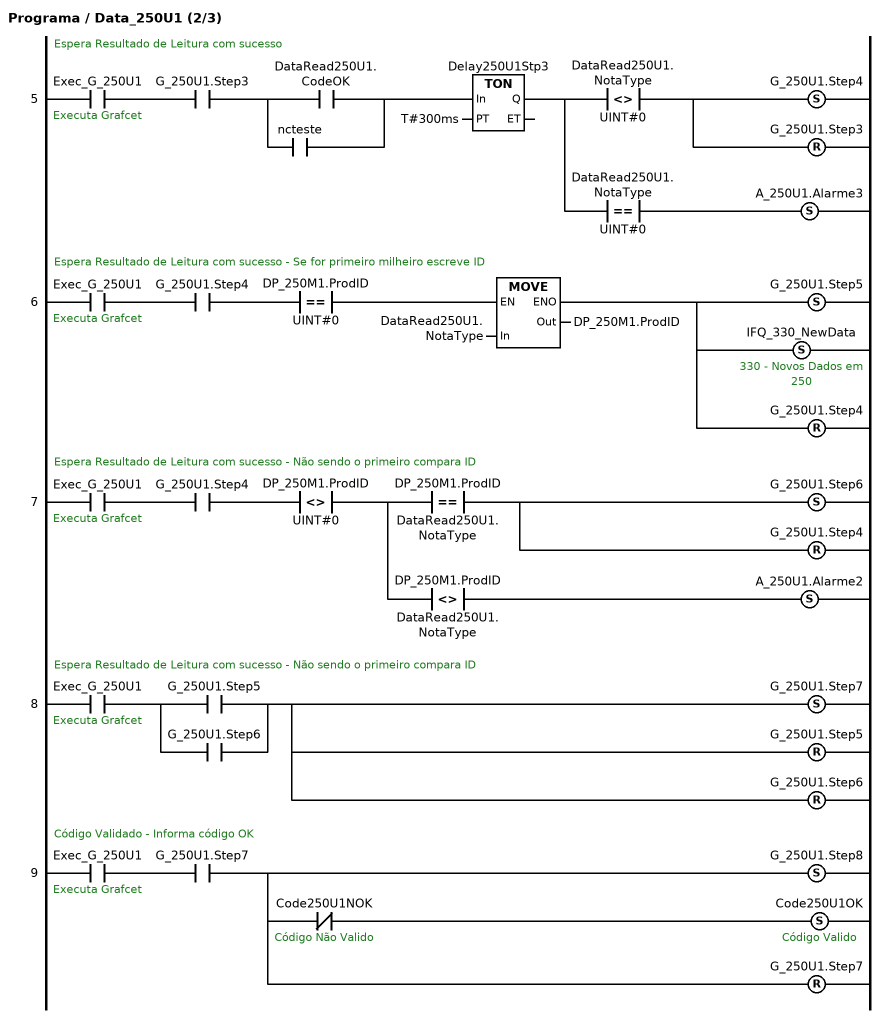
(* Rung 5: Espera Resultado de Leitura com sucesso *)
Delay250U1Stp3(In := Exec_G_250U1 AND G_250U1.Step3 AND (DataRead250U1.CodeOK OR ncteste), PT := T#300ms);
_p171 := Delay250U1Stp3.Q AND (DataRead250U1.NotaType <> UINT#0);
IF _p171 THEN
    G_250U1.Step4 := TRUE;
    G_250U1.Step3 := FALSE;
END_IF;
IF Delay250U1Stp3.Q AND (DataRead250U1.NotaType = UINT#0) THEN A_250U1.Alarme3 := TRUE; END_IF;
(* Rung 6: Espera Resultado de Leitura com sucesso - Se for primeiro milheiro escreve ID *)
_p172 := Exec_G_250U1 AND G_250U1.Step4 AND (DP_250M1.ProdID = UINT#0);
IF _p172 THEN
    DP_250M1.ProdID := DataRead250U1.NotaType;
    G_250U1.Step5 := TRUE;
    IFQ_330_NewData := TRUE;
    G_250U1.Step4 := FALSE;
END_IF;
(* Rung 7: Espera Resultado de Leitura com sucesso - Não sendo o primeiro compara ID *)
_p173 := Exec_G_250U1 AND G_250U1.Step4 AND (DP_250M1.ProdID <> UINT#0);
_p174 := _p173 AND (DP_250M1.ProdID = DataRead250U1.NotaType);
IF _p174 THEN
    G_250U1.Step6 := TRUE;
    G_250U1.Step4 := FALSE;
END_IF;
IF _p173 AND (DP_250M1.ProdID <> DataRead250U1.NotaType) THEN A_250U1.Alarme2 := TRUE; END_IF;
(* Rung 8: Espera Resultado de Leitura com sucesso - Não sendo o primeiro compara ID *)
_p175 := Exec_G_250U1 AND (G_250U1.Step5 OR G_250U1.Step6);
IF _p175 THEN
    G_250U1.Step7 := TRUE;
    G_250U1.Step5 := FALSE;
    G_250U1.Step6 := FALSE;
END_IF;
(* Rung 9: Código Validado - Informa código OK *)
_p176 := Exec_G_250U1 AND G_250U1.Step7;
IF _p176 THEN G_250U1.Step8 := TRUE; END_IF;
IF _p176 AND NOT Code250U1NOK THEN Code250U1OK := TRUE; END_IF;
IF _p176 THEN G_250U1.Step7 := FALSE; END_IF;

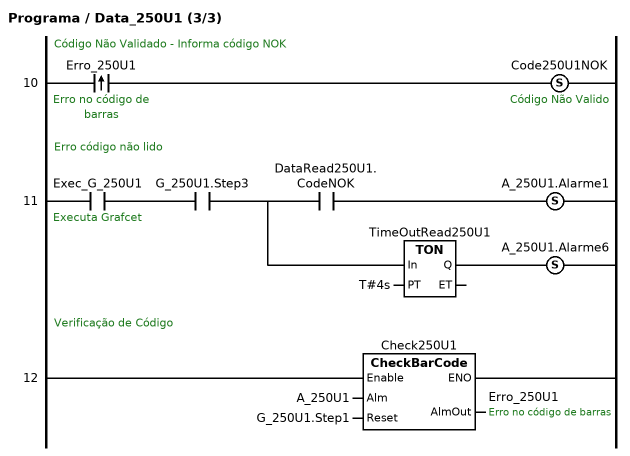
(* Rung 10: Código Não Validado - Informa código NOK *)
_e177(CLK := Erro_250U1);
IF _e177.Q THEN Code250U1NOK := TRUE; END_IF;
(* Rung 11: Erro código não lido *)
IF Exec_G_250U1 AND G_250U1.Step3 AND DataRead250U1.CodeNOK THEN A_250U1.Alarme1 := TRUE; END_IF;
TimeOutRead250U1(In := Exec_G_250U1 AND G_250U1.Step3, PT := T#4s);
IF TimeOutRead250U1.Q THEN A_250U1.Alarme6 := TRUE; END_IF;
(* Rung 12: Verificação de Código *)
Check250U1(Enable := TRUE, Alm := A_250U1, Reset := G_250U1.Step1, AlmOut => Erro_250U1);

(* Section Ctr_251V: ladder, written here as Structured Text *)

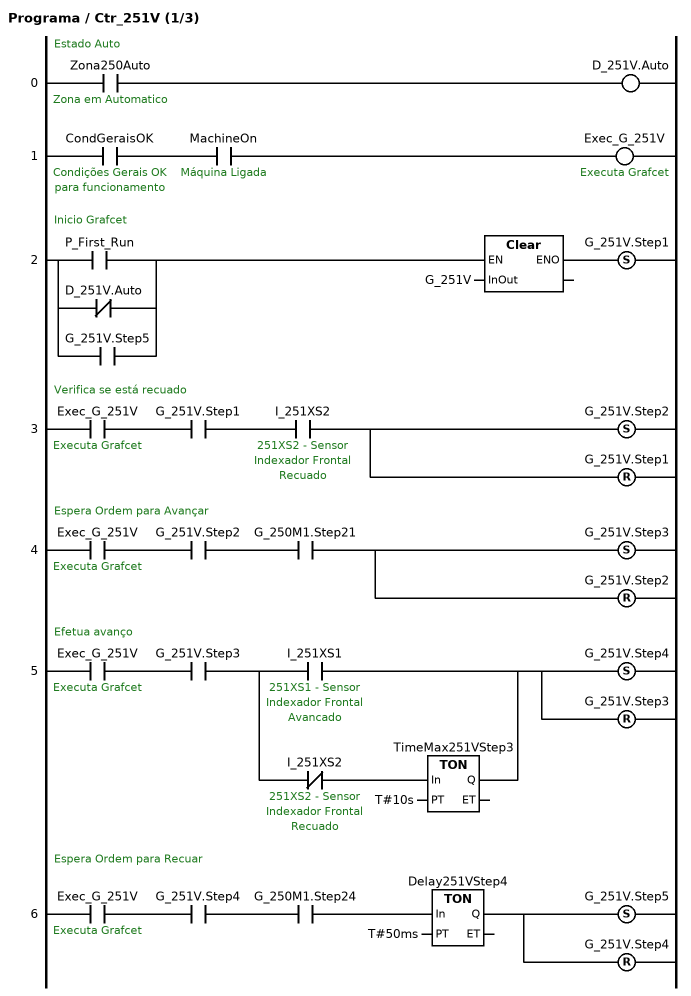
(* Rung 0: Estado Auto *)
D_251V.Auto := Zona250Auto;
(* Rung 1 *)
Exec_G_251V := CondGeraisOK AND MachineOn;
(* Rung 2: Inicio Grafcet *)
_p178 := P_First_Run OR NOT D_251V.Auto OR G_251V.Step5;
IF _p178 THEN
    Clear(InOut := G_251V);
    G_251V.Step1 := TRUE;
END_IF;
(* Rung 3: Verifica se está recuado *)
_p179 := Exec_G_251V AND G_251V.Step1 AND I_251XS2;
IF _p179 THEN
    G_251V.Step2 := TRUE;
    G_251V.Step1 := FALSE;
END_IF;
(* Rung 4: Espera Ordem para Avançar *)
_p180 := Exec_G_251V AND G_251V.Step2 AND G_250M1.Step21;
IF _p180 THEN
    G_251V.Step3 := TRUE;
    G_251V.Step2 := FALSE;
END_IF;
(* Rung 5: Efetua avanço *)
TimeMax251VStep3(In := Exec_G_251V AND G_251V.Step3 AND NOT I_251XS2, PT := T#10s);
_p181 := (Exec_G_251V AND G_251V.Step3 AND I_251XS1) OR TimeMax251VStep3.Q;
IF _p181 THEN
    G_251V.Step4 := TRUE;
    G_251V.Step3 := FALSE;
END_IF;
(* Rung 6: Espera Ordem para Recuar *)
Delay251VStep4(In := Exec_G_251V AND G_251V.Step4 AND G_250M1.Step24, PT := T#50ms);
IF Delay251VStep4.Q THEN
    G_251V.Step5 := TRUE;
    G_251V.Step4 := FALSE;
END_IF;

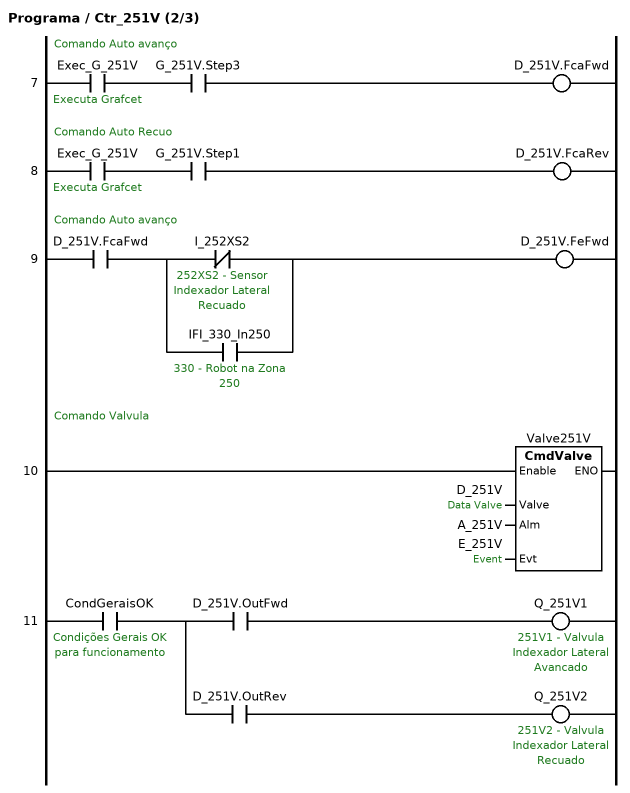
(* Rung 7: Comando Auto avanço *)
D_251V.FcaFwd := Exec_G_251V AND G_251V.Step3;
(* Rung 8: Comando Auto Recuo *)
D_251V.FcaRev := Exec_G_251V AND G_251V.Step1;
(* Rung 9: Comando Auto avanço *)
D_251V.FeFwd := D_251V.FcaFwd AND (NOT I_252XS2 OR IFI_330_In250);
(* Rung 10: Comando Valvula *)
Valve251V(Enable := TRUE, Valve := D_251V, Alm := A_251V, Evt := E_251V);
(* Rung 11 *)
Q_251V1 := CondGeraisOK AND D_251V.OutFwd;
Q_251V2 := CondGeraisOK AND D_251V.OutRev;

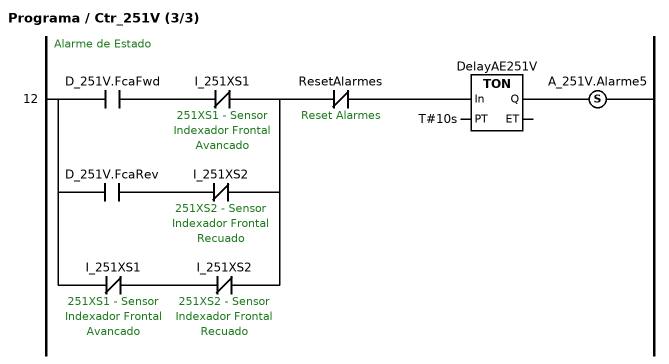
(* Rung 12: Alarme de Estado *)
DelayAE251V(In := ((D_251V.FcaFwd AND NOT I_251XS1) OR (D_251V.FcaRev AND NOT I_251XS2) OR (NOT I_251XS1 AND NOT I_251XS2)) AND NOT ResetAlarmes, PT := T#10s);
IF DelayAE251V.Q THEN A_251V.Alarme5 := TRUE; END_IF;

(* Section Ctr_252V: ladder, written here as Structured Text *)

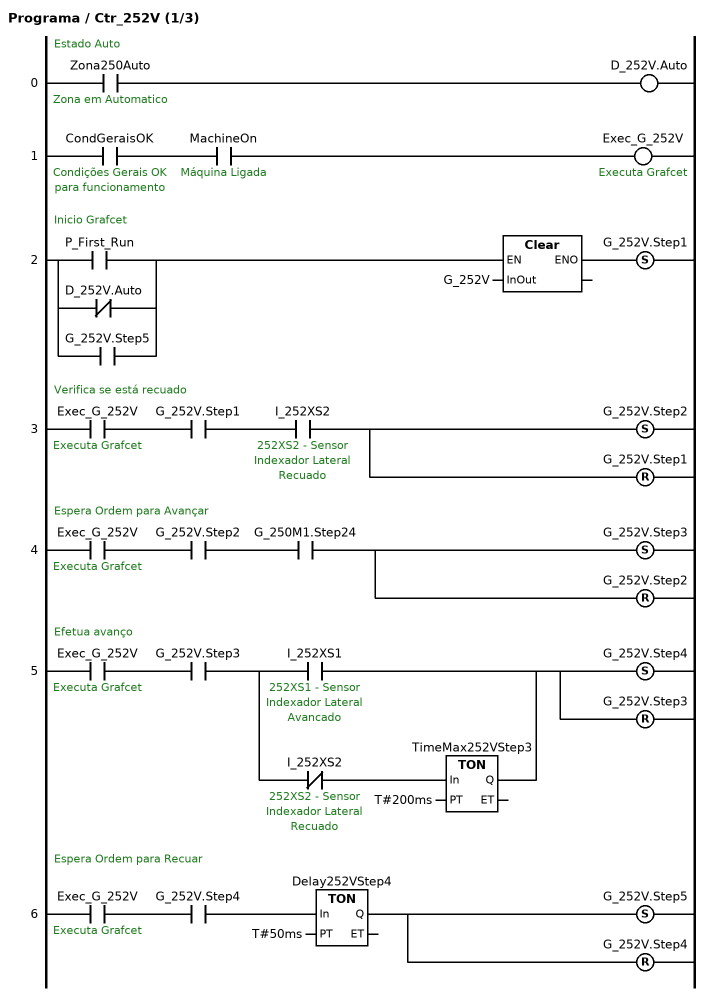
(* Rung 0: Estado Auto *)
D_252V.Auto := Zona250Auto;
(* Rung 1 *)
Exec_G_252V := CondGeraisOK AND MachineOn;
(* Rung 2: Inicio Grafcet *)
_p182 := P_First_Run OR NOT D_252V.Auto OR G_252V.Step5;
IF _p182 THEN
    Clear(InOut := G_252V);
    G_252V.Step1 := TRUE;
END_IF;
(* Rung 3: Verifica se está recuado *)
_p183 := Exec_G_252V AND G_252V.Step1 AND I_252XS2;
IF _p183 THEN
    G_252V.Step2 := TRUE;
    G_252V.Step1 := FALSE;
END_IF;
(* Rung 4: Espera Ordem para Avançar *)
_p184 := Exec_G_252V AND G_252V.Step2 AND G_250M1.Step24;
IF _p184 THEN
    G_252V.Step3 := TRUE;
    G_252V.Step2 := FALSE;
END_IF;
(* Rung 5: Efetua avanço *)
TimeMax252VStep3(In := Exec_G_252V AND G_252V.Step3 AND NOT I_252XS2, PT := T#200ms);
_p185 := (Exec_G_252V AND G_252V.Step3 AND I_252XS1) OR TimeMax252VStep3.Q;
IF _p185 THEN
    G_252V.Step4 := TRUE;
    G_252V.Step3 := FALSE;
END_IF;
(* Rung 6: Espera Ordem para Recuar *)
Delay252VStep4(In := Exec_G_252V AND G_252V.Step4, PT := T#50ms);
IF Delay252VStep4.Q THEN
    G_252V.Step5 := TRUE;
    G_252V.Step4 := FALSE;
END_IF;

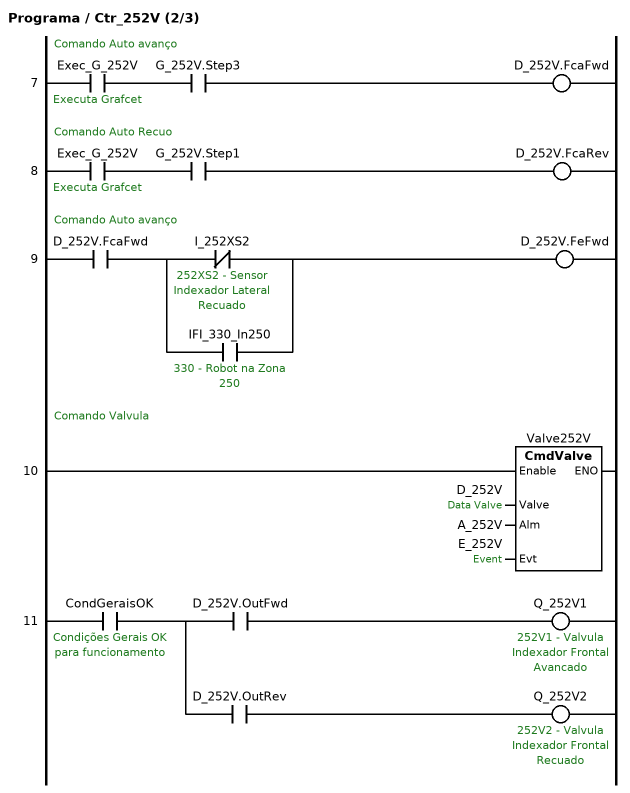
(* Rung 7: Comando Auto avanço *)
D_252V.FcaFwd := Exec_G_252V AND G_252V.Step3;
(* Rung 8: Comando Auto Recuo *)
D_252V.FcaRev := Exec_G_252V AND G_252V.Step1;
(* Rung 9: Comando Auto avanço *)
D_252V.FeFwd := D_252V.FcaFwd AND (NOT I_252XS2 OR IFI_330_In250);
(* Rung 10: Comando Valvula *)
Valve252V(Enable := TRUE, Valve := D_252V, Alm := A_252V, Evt := E_252V);
(* Rung 11 *)
Q_252V1 := CondGeraisOK AND D_252V.OutFwd;
Q_252V2 := CondGeraisOK AND D_252V.OutRev;

